FUNCTION_BLOCK ABSTRACT TcoEntity EXTENDS TcoCore.TcoObject 
VAR
    _EntityId : STRING(254);
    _Created : DATE_AND_TIME;
    _Modified : DATE_AND_TIME;
END_VAR

METHOD FB_init : BOOL
VAR_INPUT
	bInitRetains : BOOL; // if TRUE, the retain variables are initialized (warm start / cold start)
	bInCopyCode : BOOL;  // if TRUE, the instance afterwards gets moved into the copy code (online change)
	Parent : ITcoObject;
END_VAR
SUPER^.FB_init(bInitRetains := bInitRetains, bInCopyCode := bInCopyCode, Parent := Parent);
END_METHOD

END_FUNCTION_BLOCK

(* stored: Version 1.1.0.1, ProductVersion 3.1.4024.9
   POU TcoEntity: Id {6c426a5e-d492-0269-2bc4-58defc9e14b1}, SpecialFunc None
   Method FB_init: Id {19cb1922-7d5f-0097-257f-7d9b5b81e84b} *)
